// TIA Portal V16 export
// export: Created 2019-09-22T11:06:07.6180351Z, ExportSetting WithDefaults, DisplayName Totally Integrated Automation Portal, DisplayVersion V16, DisplayName TIA Portal Version Control Interface, DisplayVersion V16, DisplayName TIA Portal Openness, DisplayVersion V16, DisplayName STEP 7 Professional, DisplayVersion V16, DisplayName SIMATIC Energy Suite, DisplayVersion V16, DisplayName STEP 7 Safety, DisplayVersion V16, DisplayName WinCC Professional, DisplayVersion V16, DisplayName SIMATIC Visualization Architect, DisplayVersion V16
VAR_GLOBAL   // PLC tag table "ConstDiagnostics"
END_VAR
VAR_GLOBAL CONSTANT   // user constants
   DEV_STATE_OK : USInt := 1;   // device state ok
   DEV_STATE_LOST_CON : USInt := 3;   // device state lost connection
   DEV_STATE_DISABLED : USInt := 4;   // device state device disabled
   DEV_STATE_WAS_FAULT : USInt := 12;   // device state was fault
   DEV_STATE_WAS_LOST : USInt := 13;   // device state connection was lost
   DEV_STATE_WAS_DISABLED : USInt := 14;   // device state device was disabled
   MAX_DEVICES_SYSTEM : Int := 256;   // max number of devices per IO system
   MAX_MODULES_DEVICE : Int := 81;   // max number of modules per device
   MAX_MODULES_LOCAL : Int := 31;   // max number of local modules
   LAST_DEVICE : Int := -1;   // no next device
   MAX_SYSTEM : Int := 2;   // max number of devices per IO system
   IO_SYSTEM1 : Int := 1;   // index for IO system 1
   IO_SYSTEM2 : Int := 2;   // index for IO system 2
   IO_SYSTEM0 : Int := 0;   // index for local PLC
   DEV_STATE_FAULT : USInt := 2;   // device state fault
END_VAR
